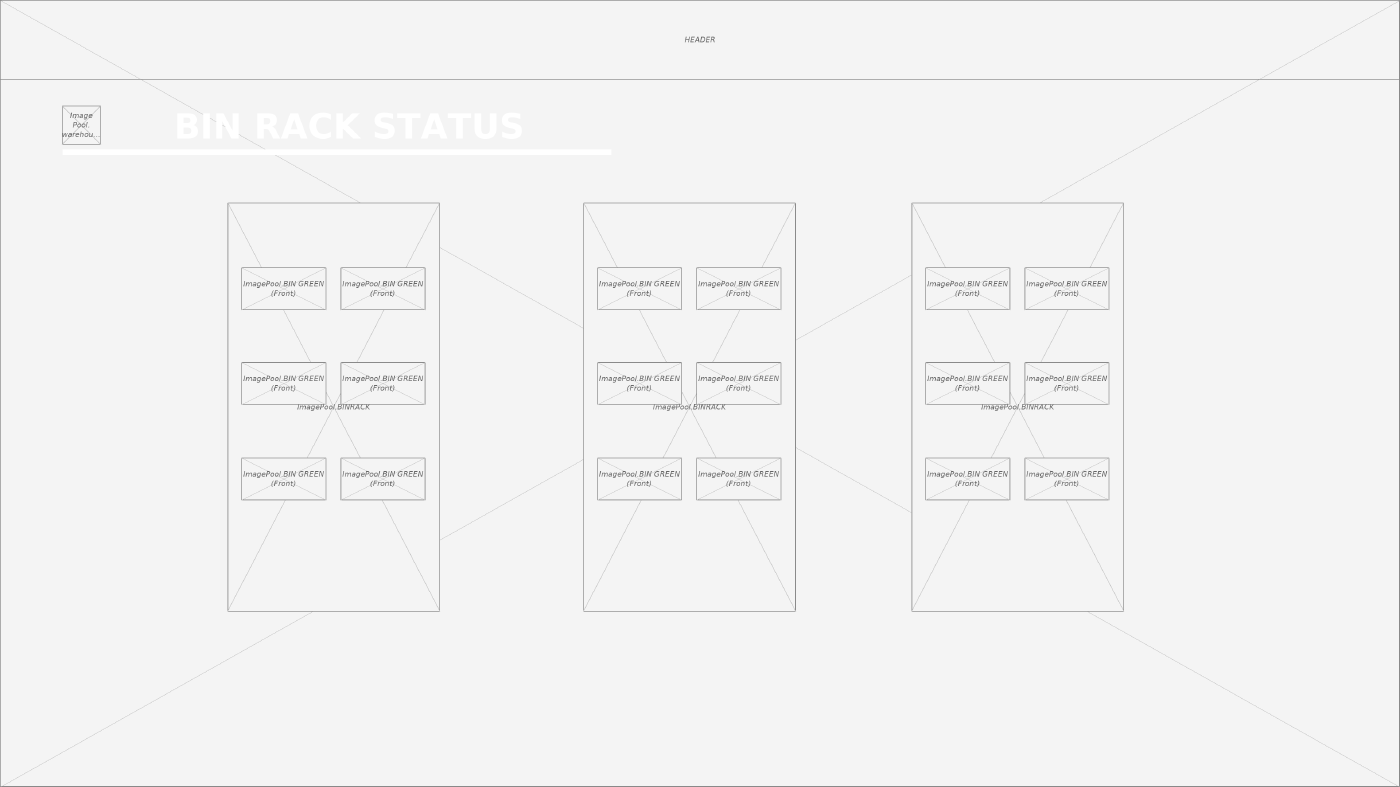
VISUALIZATION BINRACK_PAGE  // 1920x1080
    Image (0,0 1920x1080), image: ImagePool.Grey_gradient_BG
    Frame (0,0 1920x109)
        shows HEADER()
    Image (85,145 53x53), image: ImagePool.warehouse
    Rectangle (143,136 672x74), "BIN RACK STATUS"
    Rectangle (86,205 752x7)
    Group (312,278 346x668)
        Image (0,0 291x561), image: ImagePool.BINRACK
        Image (19,89 116x58), image: ImagePool.BIN GREEN (Front)
        Image (155,89 116x58), image: ImagePool.BIN GREEN (Front)
        Image (19,219 116x58), image: ImagePool.BIN GREEN (Front)
        Image (155,219 116x58), image: ImagePool.BIN GREEN (Front)
        Image (19,350 116x58), image: ImagePool.BIN GREEN (Front)
        Image (155,350 116x58), image: ImagePool.BIN GREEN (Front)
    Group (800,278 346x668)
        Image (0,0 291x561), image: ImagePool.BINRACK
        Image (19,89 116x58), image: ImagePool.BIN GREEN (Front)
        Image (155,89 116x58), image: ImagePool.BIN GREEN (Front)
        Image (19,219 116x58), image: ImagePool.BIN GREEN (Front)
        Image (155,219 116x58), image: ImagePool.BIN GREEN (Front)
        Image (19,350 116x58), image: ImagePool.BIN GREEN (Front)
        Image (155,350 116x58), image: ImagePool.BIN GREEN (Front)
    Group (1250,278 346x668)
        Image (0,0 291x561), image: ImagePool.BINRACK
        Image (19,89 116x58), image: ImagePool.BIN GREEN (Front)
        Image (155,89 116x58), image: ImagePool.BIN GREEN (Front)
        Image (19,219 116x58), image: ImagePool.BIN GREEN (Front)
        Image (155,219 116x58), image: ImagePool.BIN GREEN (Front)
        Image (19,350 116x58), image: ImagePool.BIN GREEN (Front)
        Image (155,350 116x58), image: ImagePool.BIN GREEN (Front)
END_VISUALIZATION

(* stored: Version 1.1.0.1, ProductVersion 3.1.4024.12
   Visu BINRACK_PAGE: Id {4a478f35-7f03-46e8-8a2e-1d06df070962} *)
